FUNCTION_BLOCK FB_Clock
VAR_INPUT
	TIME_ON		: TIME;	// Time to mantain clk ON
	TIME_OFF 	: TIME; // Time to mantain clk OFF
END_VAR
VAR_OUTPUT
	OUT_CLK		: BOOL; // CLK out
END_VAR
VAR
	TON_1		: TON;
	TON_2		: TON;
END_VAR

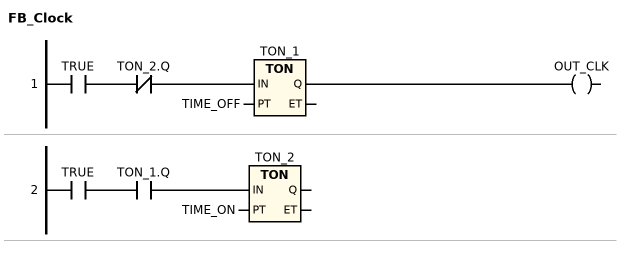
// NETWORK 1
TON_1(IN := TRUE AND NOT TON_2.Q, PT := TIME_OFF); // TON
OUT_CLK := TON_1.Q;

// NETWORK 2
TON_2(IN := TRUE AND TON_1.Q, PT := TIME_ON); // TON

END_FUNCTION_BLOCK

(* stored: Version 1.1.0.1, ProductVersion 3.1.4024.12
   POU FB_Clock: Id {972e5c9a-3f24-4afe-83a7-e898aa53a620}, SpecialFunc None *)
